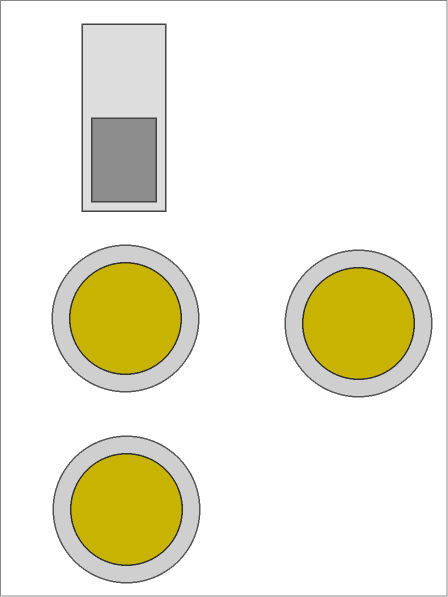
VISUALIZATION TC_VISU  // 448x597
    DipSwitch (30,18 188x199), variable: SFC_Test.Switch1, behaviour: TOGGLE, style: Switch-DipSwitch-Gray
    Lamp1 (38,233 175x171), variable: SFC_Test.Lamp1, style: Lamp-Lamp1-Yellow
    Lamp1 (39,424 175x171), variable: SFC_Test.Lamp2, style: Lamp-Lamp1-Yellow
    Lamp1 (271,238 175x171), variable: SFC_Test.Lamp3, style: Lamp-Lamp1-Yellow
END_VISUALIZATION

(* stored: Version 1.1.0.1, ProductVersion 3.1.4022.10
   Visu TC_VISU: Id {f945a80b-bdea-4889-87c3-0cfd965e94f9} *)
